{attribute 'qualified_only'}
{attribute 'strict'}
(*
	Structure used to couple limit switches of slaves to master axes
*)
TYPE eLimitCoupling :
(
	None,
	FwSw,
	BwSw,
	Both	//not implemented
);
END_TYPE

(* stored: Version 1.1.0.1, ProductVersion 3.1.4022.12
   DUT eLimitCoupling: Id {7810a9bc-d383-47ea-8dc8-4d10bb134045} *)
